// TIA Portal V18 export
TYPE "LGasp_typeTracking"
// stored: IsFailsafeCompliant false
   STRUCT
      nome_stz : String["NumCharTrackingStazione"];   // nome stazione
      en_reset : Bool;   // abilita reset posizione tracking
      state : Int;   // stato stazione
      info : "LGasp_typeTrackingPart";
   END_STRUCT;
END_TYPE
